# B&R Automation Studio project Soiled_PLC (part 19)

#### Main.st - Init, cyclic, exit code
```iecst
//V2.00.1 -- First stable release
//V2.00.2 -- Set brake control to be optional - This means changing when we encode the paramater structure.
//V2.00.3 -- Add new constant to set MAX_FREQUENCY
//V2.00.4 -- If the drive started not on remote it wouldn;t always go into config to start. ADD new mode for when module ok is false.
//V2.00.5 -- Add test mode for simulation
//V2.00.6 -- BUG FIX -- Minumum speed was being set to Max which stopped speed control
//V2.00.7 -- REMOVE -- Remove the old structure for settings via http
//V2.00.8 -- FIX -- Correct the scaling of MaxCurrent from settings - we now us 200 = 2A
PROGRAM _INIT
	FOR n := 1 TO MAX_DRIVES DO
		drive ACCESS ADR(ABB_EPL.Drives[n]);
		drive.Cmd.Node := 100 + n; //Set node here for now, may move to belt task
		drive.Comm.State := ABB_CONFIG;
		drive.Config.currentParam := 1; //Reset starting parameter index
	END_FOR;
END_PROGRAM

PROGRAM _CYCLIC

	FOR n := 1 TO MAX_DRIVES DO
		IF (testDrive > 0) THEN
			drive ACCESS ADR(ABB_EPL.Drives[testDrive]);
		ELSE
			drive ACCESS ADR(ABB_EPL.Drives[n]);
		END_IF;

		//Control Word												Status Word
		//Bit 0		Switch On										Bit 0	Ready To Switch On
		//Bit 1		Enable Voltage									Bit 1	Switched On
		//Bit 2		Quick Stop										Bit 2	Operation Enabled
		//Bit 3		Enable Operation								Bit 3	Fault
		//Bit 4		Not Used In Scalor Mode							Bit 4	Voltage Enabled
		//Bit 5		Not Used In Scalor Mode							Bit 5	Quick Stop
		//Bit 6		Not Used In Scalor Mode							Bit 6	Switch On Disabled
		//Bit 7		Fault Reset										Bit 7 	Warning
		//Bit 8		Halt											Bit 8	Drive Specific TBC
		//Bit 9		Operation Mode Specific							Bit 9	Remote
		//Bit 10	Reserved	??Remote Control??					Bit 10	Target Reached
		//Bit 11	Drive Specific	TBC								Bit 11 	Internal Limit Reached
		//Bit 12	Drive Specific	TBC								Bit 12	Not Used In Scalor Mode
		//Bit 13	Drive Specific	TBC								Bit 13	Not Used In Scalor Mode
		//Bit 14	Drive Specific	TBC								Bit 14	Drive Specific TBC
		//Bit 15	Drive Specific	TBC								Bit 15	Drive Specific TBC

		//Use a local instance of controlword so we don't pass changing data to the drive while processing

		controlWord := SHUT_DOWN;	// 0000 0000 0111 0110

		//Encode the controlword and statusword
		abb_packData(pData := ADR(drive));
		IF TestSystem AND NOT drive.Comm.ModuleOk THEN // TEST MODE
			IF drive.Cmd.Run THEN
				drive.Comm.State := ABB_RUNNING;
			ELSE
				drive.Status.ReadyToRun := 1;
			END_IF;
		ELSIF NOT drive.Comm.ModuleOk THEN
			drive.Comm.State := ABB_DISCONNECTED;
		ELSIF (drive.Config.params[MAX_PARAMS].status <> 0) OR (drive.Config.currentParam < MAX_PARAMS) THEN
			drive.Comm.State := ABB_CONFIG;
		ELSIF NOT drive.Status.OnRemote THEN
			drive.Comm.State := ABB_OFF_REMOTE;
		ELSIF drive.Status.Tripped THEN
			drive.Comm.State := ABB_TRIPPED;
		ELSIF NOT drive.Cmd.QuickStop THEN	//Enable quick stop
			drive.Comm.State := ABB_QUICK_STOP;
		ELSIF drive.Status.SwitchOnInhibit THEN
			drive.Comm.State := ABB_SWITCH_ON_INHIBITED;
		ELSIF drive.Comm.ErrorCode = ABB_FAULT_STO THEN
			drive.Comm.State := ABB_STO;
		END_IF;

		CASE drive.Comm.State OF

			ABB_DISCONNECTED:
				drive.Config.currentParam := 1; // Force write of parameters

			ABB_CONFIG: //Wait for module OK to be TRUE
				_setParameters; //Write params
				IF drive.Comm.ModuleOk AND (drive.Config.params[MAX_PARAMS].status = 0) THEN
					drive.Comm.State := ABB_SWITCH_ON_INHIBITED;
				END_IF;

			ABB_SWITCH_ON_INHIBITED:	//Wait for quick stop and enable to be true
				IF NOT drive.Status.SwitchOnInhibit THEN
					drive.Comm.State := ABB_NOT_READY_TO_SWITCH_ON;
				END_IF;

			ABB_NOT_READY_TO_SWITCH_ON:
				IF drive.Status.ReadyToSwitchOn THEN
					drive.Comm.State := ABB_READY_TO_SWITCH_ON;
				END_IF;

			ABB_READY_TO_SWITCH_ON:
				controlWord := SWITCH_ON; //0000 0111 0111
				IF drive.Status.ReadyToRun THEN
					drive.Comm.State := ABB_READY_TO_RUN;
				END_IF;

			ABB_READY_TO_RUN:
				controlWord := SWITCH_ON; //0000 0111 0111
				IF drive.Cmd.Run AND (ABS(drive.Cmd.TargetVelocity) >= ABB_MIN_VELOCITY) THEN	//Check min frequency is met
					drive.Comm.State := ABB_RUNNING;
				END_IF;

			ABB_RUNNING:
				controlWord := ENABLE_OPERATION; //0000 0111 1111

				IF NOT drive.Cmd.Run THEN
					drive.Comm.State := ABB_RAMP_DOWN;
				END_IF;

			ABB_RAMP_DOWN:
				controlWord := RAMP_DOWN; //0001 0111 1111
				IF drive.Comm.StatusWord.11 = 0 AND drive.Comm.ActVelocity = 0 THEN
					drive.Comm.State := ABB_READY_TO_RUN;
				END_IF;

			ABB_QUICK_STOP:
				controlWord := QUICK_STOP; //0000 0111 0010
				IF drive.Comm.StatusWord.11 = 0 AND drive.Comm.ActVelocity = 0 AND drive.Cmd.QuickStop THEN
					drive.Comm.State := ABB_READY_TO_RUN;
				END_IF;

			ABB_TRIPPED:
				//We must wait for the drive to be ready for reset and give an edge..
				controlWord := DISABLE_VOLTAGE; //0000 0000 0000
				IF drive.Comm.StatusWord.11 = 0 AND drive.Comm.ActVelocity = 0 AND NOT drive.Cmd.Reset THEN //Toggle reset to generate edge
					controlWord := FAULT_RESET;
					drive.Cmd.Reset := TRUE;
				ELSE
					drive.Cmd.Reset := FALSE;
				END_IF;
				//We can auto reset here..but we should log an error somewhere..
				IF NOT drive.Status.Tripped THEN
					drive.Comm.State := ABB_SWITCH_ON_INHIBITED;
				END_IF;

			ABB_OFF_REMOTE:
				//Remote control not active
				controlWord := SET_REMOTE;
			////				IF drive.Status.OnRemote THEN
			////					IF (drive.Config.params[MAX_PARAMS].status <> 0) THEN
			////						drive.Comm.State := ABB_CONFIG;
			////					ELSE
			////						drive.Comm.State := ABB_SWITCH_ON_INHIBITED;
			////					END_IF;
			////				END_IF;
			//				IF NOT Std.Drives_AllowLocalMode AND (drive.Config.params[13].data = Std.Drives_AllowLocalMode) THEN //Only reset the parameters if the local control mode has chnaged
			//					_encodeParameters;
			//					drive.Config.currentParam := 1; //Reset starting parameter index
			//				END_IF;
			//
			ABB_STO:
				IF drive.Comm.ErrorCode <> ABB_FAULT_STO THEN
					drive.Comm.State := ABB_SWITCH_ON_INHIBITED;
				END_IF;
		END_CASE;
		drive.Status.Running := (drive.Comm.State =  ABB_RUNNING);
		drive.Comm.ControlWord := controlWord;
	END_FOR;

	//Temp code so that we can set a node number, The NODE must already be set to 1 (DEFAULT)
	IF (newNode > 0) THEN
		setNodeNumber.enable := 1;
		setNodeNumber.node := 1;
		setNodeNumber.index := 16#4033;
		setNodeNumber.subindex := 16#03;
		setNodeNumber.pData :=  ADR(newNode);
		setNodeNumber.datalen := 2;
		setNodeNumber();
		IF (setNodeNumber.status = ERR_OK) THEN
			newNode := 0;
		END_IF;
	ELSIF saveNewNode THEN
		saveVar := 1;
		setNodeNumber.enable := 1;
		setNodeNumber.node := 1;
		setNodeNumber.index := 16#4033;
		setNodeNumber.subindex := 16#1B;
		setNodeNumber.pData :=  ADR(saveVar);
		setNodeNumber.datalen := 2;
		setNodeNumber();
		IF (setNodeNumber.status = ERR_OK) THEN
			saveNewNode := 0;
		END_IF;
	ELSIF (factoryReset > 0) THEN
		saveVar := 34560;
		setNodeNumber.enable := 1;
		setNodeNumber.node := UINT_TO_USINT(factoryReset);
		setNodeNumber.index := 16#4060;
		setNodeNumber.subindex := 16#06;
		setNodeNumber.pData :=  ADR(saveVar);
		setNodeNumber.datalen := 2;
		setNodeNumber();
		IF (setNodeNumber.status = ERR_OK) THEN
			factoryReset := 0;
		END_IF;
	END_IF;

END_PROGRAM
```

#### Types.typ - Local data types
```iecst
TYPE
	state_enum :
		(
		SLOW := 0,
		FAST := 1,
		ACC := 2,
		DEC := 3,
		MAXCURRENT := 4
		);
	BackUp : 	STRUCT
		filePath : STRING[15];
		fileDevice : STRING[10];
		status : UINT;
		ident : UDINT;
		step : backUp_enum;
		functions : backUp_functions;
	END_STRUCT;
	backUp_enum :
		(
		backUpStart := 0,
		backUpOpen := 1,
		backUpCreate := 2,
		backUpWrite := 3,
		backUpRead := 4,
		backUpClose := 5,
		backUpErrorRead := 6,
		backUpErrorWrite := 7,
		backUpExit := 100
		);
	backUp_functions : 	STRUCT
		fWrite : FileWrite;
		fRead : FileRead;
		fOpen : FileOpen;
		fCreate : FileCreate;
		fClose : FileClose;
	END_STRUCT;
END_TYPE
```

#### Variables.var - Local variables
```iecst
VAR
	abb_packData : ABB_PackData; (*Decodes status word and encodes some parameters*)
	drive : REFERENCE TO ABB_EPL_typ; (*ref var to drive structure*)
	controlWord : UINT; (*control word for drive*)
	n : USINT; (*used to hold loop state*)
	write : REFERENCE TO ABB_EPL_Param_Write_typ; (*ref var to write structutre within drive structure*)
	testDrive : UINT; (*set this to drive number you want to test*)
	i : USINT;
	state : state_enum;
	count : USINT;
	test : UINT;
	newNode : UINT;
	saveNewNode : BOOL;
	saveVar : UINT;
	factoryReset : UINT;
	setNodeNumber : EplSDOWrite;
END_VAR
```

#### encodeParameters.st
```iecst
//-----------------------------------------
//--AsEPL library Status Error Codes-------
//-----------------------------------------

//Error									Description
//0  										No error
//65534  								Function block parameter "enable" not equal to 1
//65535  								Function block still working

//31340  								Basis of error numbers, internal error
//31341  								Specified device not a POWERLINK interface
//31342  								Function can only be executed on an MN (managing node).
//31343  								Function can only be executed on a CN (controlled node).
//31344  								Read or write access failed. See errorinfo for the precise cause of the error.
//31345  								Input parameters outside of permitted value range
//31346  								Specified index already exists
//31347  								Specified subindex already exists
//31348  								Specified index does not exist
//31349  								Specified subindex does not exist
//31392  								Null pointer given as data buffer
//31399  								Error code for non-implemented functionality

//-----------------------------------------
//-----AsEPL library Error Info Codes------
//-----------------------------------------

//Error									Description
//16#0504_0000 					SDO communication timeout.
//16#0504_0001 					Invalid or unknown client/server command.
//16#0504_0002 					Size of transferred data invalid.
//16#0504_0003 					Error in sequence layer.
//16#0504_0005 					Could not allocate enough memory.
//16#0601_0000 					Cannot access object.
//16#0601_0001 					Attempted to read a write-only object.
//16#0601_0002 					Attempted to write a read-only object.
//16#0602_0000 					Object not in object dictionary.
//16#0604_0041 					Attempted to map an object in the PDO that doesn't support it.
//16#0604_0042 					Assignment would exceed PDO length.
//16#0604_0043 					General parameter incompatibility.
//16#0604_0047 					General device incompatibility.
//16#0606_0000 					Access failed due to hardware error.
//16#0607_0010 					Data type doesn't match the length of the access.
//16#0607_0012 					Length of the access is larger than the length of the data type.
//16#0607_0013 					Length of the access is smaller than the length of the data type.
//16#0609_0011 					Subindex does not exist.
//16#0609_0030 					Invalid value range.
//16#0609_0031 					Value too high for value range.
//16#0609_0032 					Value too low for value range.
//16#0609_0036 					Maximum value less than minimum value.
//16#0800_0000 					General error.
//16#0800_0020 					Cannot transfer or store data.
//16#0800_0021 					Data cannot be transferred or stored since it's being used locally by the device.
//16#0800_0022 					Data cannot be transferred or saved due to the device state.

ACTION _encodeParameters:
	//Clear all parameters
	FOR i:= 1 TO MAX_PARAMS DO
		//Clear stauts/error
		drive.Config.params[i].status := 1; //Set to 1 here, if not cleared when written is shows it has not been written
		drive.Config.params[i].errorInfo := 0;
	END_FOR;

	//Set all parameters
	//Brake Function
	drive.Config.params[1].index := 16#402C;	//Brake Control Enable 44.06
	drive.Config.params[1].subIndex := 16#6;
	drive.Config.params[1].data := BOOL_TO_DINT(drive.Cmd.BrakeFitted);	//Enable brake control
	drive.Config.params[1].datalen := 4;

	drive.Config.params[2].index := 16#400A;	//RO1 Source 10.24
	drive.Config.params[2].subIndex := 16#18;
	drive.Config.params[2].data := 22;	//Relay is active when brake is active
	drive.Config.params[2].datalen := 4;

	//Motor Data
	drive.Config.params[3].index := 16#4063;	//Motor Nominal Voltage 99.07
	drive.Config.params[3].subIndex := 16#7;
	drive.Config.params[3].data := 4150;	//415V
	drive.Config.params[3].datalen := 4;

	drive.Config.params[4].index := 16#4063;	//Motor Nominal Frequency 99.08
	drive.Config.params[4].subIndex := 16#8;
	drive.Config.params[4].data := 5000;	//50Hz
	drive.Config.params[4].datalen := 4;

	drive.Config.params[5].index := 16#4063;	//Motor Power Factor 99.11
	drive.Config.params[5].subIndex := 16#B;
	drive.Config.params[5].data := 80;	//0.8
	drive.Config.params[5].datalen := 4;

	drive.Config.params[6].index := 16#4063;	//Motor Control Mode 99.04
	drive.Config.params[6].subIndex := 16#4;
	drive.Config.params[6].data := 1;	//Scalor
	drive.Config.params[6].datalen := 2;

	//Limits
	drive.Config.params[7].index := 16#401E;	//Max Current 30.17
	drive.Config.params[7].subIndex := 16#11;
	drive.Config.params[7].data := 200;	//2.0A
	drive.Config.params[7].datalen := 4;

	drive.Config.params[8].index := 16#401E;	//Max Frequency 30.14
	drive.Config.params[8].subIndex := 16#E;
	drive.Config.params[8].data := MAX_FREQUENCY_HZ * 100;	//60Hz
	drive.Config.params[8].datalen := 4;

	//Fault Functions
	//	drive.Config.params[9].index := 16#401F;	//External Event 1 Source 31.01
	//	drive.Config.params[9].subIndex := 16#1;
	//	drive.Config.params[9].data := 2;	//Digital Input 1 Triggers Fault When Low
	//	drive.Config.params[9].datalen := 4;

	drive.Config.params[9].index := 16#4032;	//Comms loss function 50.02
	drive.Config.params[9].subIndex := 16#2;
	drive.Config.params[9].data := 1;	//Fault on comms loss
	drive.Config.params[9].datalen := 2;

	//Other
	drive.Config.params[10].index := 16#4014;	//External Commands 20.01
	drive.Config.params[10].subIndex := 16#1;
	drive.Config.params[10].data := 12;	//Fieldbus A Selected
	drive.Config.params[10].datalen := 2;

	drive.Config.params[11].index := 16#401C;	//Frequency Ext 1 Ref 28.11
	drive.Config.params[11].subIndex := 16#B;
	drive.Config.params[11].data := 4;	//Fieldbus A As Ref
	drive.Config.params[11].datalen := 4;

	drive.Config.params[12].index := 16#401F;	//STO Indication 31.22
	drive.Config.params[12].subIndex := 16#16;
	drive.Config.params[12].data := 3;	//Warning/Warning
	drive.Config.params[12].datalen := 2;

	drive.Config.params[13].index := 16#4013;	//Disable local mode 19.17
	drive.Config.params[13].subIndex := 16#11;
	drive.Config.params[13].data := BOOL_TO_DINT(NOT Std.Drives_AllowLocalMode);// 0 = Enabled ,1 = Locked
	drive.Config.params[13].datalen := 2;

	drive.Config.params[14].index := 16#4032;	//Comm loss time out 50.03
	drive.Config.params[14].subIndex := 16#3;
	drive.Config.params[14].data := 15;	//1 second
	drive.Config.params[14].datalen := 2;

	drive.Config.params[15].index := 16#401E;	//Min Frequency 30.13
	drive.Config.params[15].subIndex := 16#D;
	drive.Config.params[15].data := MAX_FREQUENCY_HZ * -100;
	drive.Config.params[15].datalen := 4;

END_ACTION
```

#### setParameters.st
```iecst
ACTION _setParameters:
	//V2.00.2 Encode parameters
	_encodeParameters;

	//Overwrite Max current
	IF ABB_EPL.Settings[drive.Cmd.Node-100].MaxCurrent > 0 THEN
		drive.Config.params[7].data := ABB_EPL.Settings[drive.Cmd.Node-100].MaxCurrent;
	END_IF;
	drive.Cmd.Acc_seconds := ABB_EPL.Settings[drive.Cmd.Node-100].Acc;
	drive.Cmd.Dec_seconds := ABB_EPL.Settings[drive.Cmd.Node-100].Dec;

	drive.Config.function.enable := TRUE;																	//Enable function block
	drive.Config.function.pDevice := ADR(PLK_INTERFACE);														//Set powerlink address in ABB_Driver init task
	drive.Config.function.node := drive.Cmd.Node; 															//Node number of drive, set in ABB_EPL[n].cmd.node if non standard.

	IF drive.Config.currentParam <= MAX_PARAMS THEN
		IF (drive.Config.params[drive.Config.currentParam].status > 0) THEN									//Call function only if not completed
			drive.Config.function.index := drive.Config.params[drive.Config.currentParam].index; 			//Powerlink index address
			drive.Config.function.subindex := drive.Config.params[drive.Config.currentParam].subIndex;		//Powerlink sub index address
			drive.Config.function.pData := ADR(drive.Config.params[drive.Config.currentParam].data);		//Value of data to write
			drive.Config.function.datalen := drive.Config.params[drive.Config.currentParam].datalen;		//Size of data type														//Call function
			IF (drive.Config.function.status = ERR_OK) THEN 												//Clear errors
				drive.Config.params[drive.Config.currentParam].status := 0;
				drive.Config.params[drive.Config.currentParam].errorInfo := 0;
				drive.Config.currentParam := drive.Config.currentParam + 1;
			ELSIF (drive.Config.function.status <> ERR_FUB_BUSY) AND (drive.Config.function.status <> ERR_FUB_ENABLE_FALSE) THEN //Store errors
				drive.Config.params[drive.Config.currentParam].status := drive.Config.function.status;
				drive.Config.params[drive.Config.currentParam].errorInfo := drive.Config.function.errorinfo;
				drive.Config.function.enable := FALSE;
//			ELSIF drive.Config.function.status <> 20925 THEN;//ERR_PLMGR_STATION_NOT_ACTIVE THEN  //Only skip if the devuce is active																																					//Skip if other error to stop PLC hanging in bootup
//				drive.Config.params[drive.Config.currentParam].status := drive.Config.function.status;
//				drive.Config.params[drive.Config.currentParam].errorInfo := drive.Config.function.errorinfo;
//				drive.Config.currentParam := drive.Config.currentParam + 1;
			END_IF;
			drive.Config.function();
		ELSE
			drive.Config.function.enable := FALSE;
		END_IF;
	END_IF;

	//Parameters should be loaded onto default settings.
	//to default the drive set 9606 t0 34560
	//Node ID (5103) has to be manually set

	write ACCESS ADR (drive.Parameters.Write);

	CASE drive.Cmd.MotorSize OF // Need to set these values correctly

		ABB_MOTOR_0_25KW:
			write.Motor_NominalCurrent_9906		:= 7; //0.68 A
			write.Motor_NominalPower_9910		:= 25; // 0.37 kW
			write.Motor_NominalSpeed_9909 		:= 1300;

		ABB_MOTOR_0_37KW_0_91A_1374:
			write.Motor_NominalCurrent_9906		:= 9; //0.91 A
			write.Motor_NominalPower_9910		:= 37; // 0.37 kW
			write.Motor_NominalSpeed_9909 		:= 1374;

		ABB_MOTOR_0_37KW_0_97A_1342:
			write.Motor_NominalCurrent_9906		:= 10; //0.97 A
			write.Motor_NominalPower_9910		:= 37; // 0.37 kW
			write.Motor_NominalSpeed_9909 		:= 1342;

		ABB_MOTOR_0_37KW_1_14A_1380:
			write.Motor_NominalCurrent_9906		:= 7; //1.14 A
			write.Motor_NominalPower_9910		:= 37; // 0.37 kW
			write.Motor_NominalSpeed_9909 		:= 1380;

		ABB_MOTOR_0_75KW:
			write.Motor_NominalCurrent_9906		:= 18; //1.75 A
			write.Motor_NominalPower_9910		:= 75; // 0.75 kW
			write.Motor_NominalSpeed_9909 		:= 1440;

		ABB_MOTOR_1_5KW:
			write.Motor_NominalCurrent_9906		:= 30;// 3 A?
			write.Motor_NominalPower_9910		:= 150;// 1.5kW
			write.Motor_NominalSpeed_9909 		:= 1450;

		ABB_MOTOR_2_2KW_4_75A_1450:
			write.Motor_NominalCurrent_9906		:= 48; //4.75 A
			write.Motor_NominalPower_9910		:= 220; // 2.2 kW
			write.Motor_NominalSpeed_9909 		:= 1450;

		ABB_MOTOR_3KW:
			write.Motor_NominalCurrent_9906		:= 64;
			write.Motor_NominalPower_9910		:= 300; // 3 kW
			write.Motor_NominalSpeed_9909 		:= 1456;

		ABB_MOTOR_CUSTOM: // Future  Alow Motor data to be set individaully
		//write.Motor_NominalCurrent_9906		:= 100;
		//write.Motor_NominalPower_9910			:= ;
		//write.Motor_NominalSpeed_9909 		:= 1450; //RPM
		//Over current = ??
		//Over torque = ??

	END_CASE;
END_ACTION
```

### Library Logical/ABB_EPL/ABB_EPL (IEC)
Depends on: AsEPL

#### ABB_EPL.typ
```iecst
TYPE
	ABB_Settings_typ : 	STRUCT
		Slow : INT;
		Fast : INT;
		Acc : INT; (*This is passed back as a whole number to make decoding easier. This in milli seconds and must be /1000 and cast to REAL.*)
		Dec : INT; (*This is passed back as a whole number to make decoding easier. This in milli seconds and must be /1000 and cast to REAL.*)
		MaxCurrent : DINT;
	END_STRUCT;
	ABB_EPL_Struct : 	STRUCT
		Settings : ARRAY[1..MAX_DRIVES]OF ABB_Settings_typ;
		Drives : ARRAY[1..MAX_DRIVES]OF ABB_EPL_typ;
		httpRequest : STRING[5000];
		httpResponse : ARRAY[0..4999]OF USINT;
		callBackUpWrite : BOOL;
	END_STRUCT;
	ABB_EPL_typ : 	STRUCT
		Comm : ABB_EPL_Comm_typ;
		Cmd : ABB_EPL_cmd_typ;
		Status : ABB_EPL_status_typ;
		Parameters : ABB_EPL_Param_typ;
		Config : EPL_Config;
	END_STRUCT;
	ABB_EPL_Comm_typ : 	STRUCT
		ControlWord : UINT;
		StatusWord : UINT;
		TargetVelocity : INT; (*RPM*)
		ActVelocity : INT; (*RPM*)
		ModuleOk : BOOL;
		State : ABB_EPL_Comm_State_enum;
		ActCurrent : DINT;
		ActTorque : DINT;
		ErrorCode : UINT;
	END_STRUCT;
	ABB_Motor_Size_enum :
		(
		ABB_MOTOR_0_25KW,
		ABB_MOTOR_0_37KW_0_91A_1374,
		ABB_MOTOR_0_37KW_0_97A_1342,
		ABB_MOTOR_0_37KW_1_14A_1380,
		ABB_MOTOR_0_75KW,
		ABB_MOTOR_1_5KW,
		ABB_MOTOR_2_2KW_4_75A_1450,
		ABB_MOTOR_3KW,
		ABB_MOTOR_CUSTOM
		);
	ABB_EPL_cmd_typ : 	STRUCT
		TargetVelocity : INT; (*RPM*)
		Run : BOOL;
		Reset : BOOL;
		QuickStop : BOOL;
		MotorSize : ABB_Motor_Size_enum;
		Dec_seconds : REAL; (*Decleration Time Seconds*)
		Acc_seconds : REAL; (*Acceleration Time Seconds*)
		Direction : ABB_DIRECTION_Enum;
		Node : USINT; (*Powerlink Node Address*)
		BrakeFitted : BOOL; (*Does the motor have a brake fitted*)
	END_STRUCT;
	ABB_EPL_status_typ : 	STRUCT
		ReadyToSwitchOn : BOOL;
		ReadyToRun : BOOL;
		Tripped : BOOL;
		DriveEnabled : BOOL;
		QuickstopActive : BOOL;
		SwitchOnInhibit : BOOL;
		Warning : BOOL;
		AtSpeed : BOOL; (**Drive is running at target velocity*)
		ActCurrent : DINT; (*Amps*)
		ActTorque : DINT; (*% of nominal motor torque*)
		ThermalTrip : BOOL;
		OnRemote : BOOL; (**Powerlink control is active*)
		Running : BOOL;
	END_STRUCT;
	ABB_EPL_Comm_State_enum :
		(
		ABB_DISCONNECTED,
		ABB_QUICK_STOP,
		ABB_CONFIG,
		ABB_SWITCH_ON_INHIBITED,
		ABB_NOT_READY_TO_SWITCH_ON,
		ABB_READY_TO_SWITCH_ON,
		ABB_READY_TO_RUN,
		ABB_RUNNING,
		ABB_TRIPPED,
		ABB_OFF_REMOTE, (**Drive not on remote control*)
		ABB_STO,
		ABB_RAMP_DOWN
		);
	ABB_EPL_Param_typ : 	STRUCT
		Read : ABB_EPL_Param_Read_typ;
		Write : ABB_EPL_Param_Write_typ;
	END_STRUCT;
	ABB_EPL_Param_Read_typ : 	STRUCT
		ActCurrent_0107 : DINT; (*Amps*)
		ActTorque_0110 : DINT; (*% of nominal motor torque*)
	END_STRUCT;
	ABB_EPL_Param_Write_typ : 	STRUCT
		Ramp_AccTime1_2872 : DINT;
		Ramp_DecTime1_2873 : DINT;
		Motor_NominalCurrent_9906 : DINT; (*1=1A*)
		Motor_NominalSpeed_9909 : DINT; (*Nominal Speed RPM*)
		Motor_NominalPower_9910 : DINT;
		QuickStopTime_2323 : DINT; (*Time in seconds for emergency stop*)
	END_STRUCT;
	ABB_DIRECTION_Enum :
		(
		ABB_DIRECTION_FWD,
		ABB_DIRECTION_REV
		);
	EPL_Config : 	STRUCT
		function : EplSDOWrite;
		currentParam : USINT;
		New_Member : USINT;
		params : ARRAY[0..MAX_PARAMS]OF EPL_SDO;
	END_STRUCT;
	EPL_SDO : 	STRUCT
		index : UINT;
		subIndex : USINT;
		data : DINT;
		datalen : UDINT;
		status : UINT;
		errorInfo : UDINT;
	END_STRUCT;
END_TYPE
```

#### Config.var
```iecst
VAR CONSTANT
	MAX_DRIVES : USINT := 23; (*Set to number of drives*)
	MAX_FREQUENCY_HZ : USINT := 70; (*Maximum Frequency Allowed in hz*)
	ABB_MIN_VELOCITY : USINT := 20; (*Minimum allowable speed of the drive*)
	PLK_INTERFACE : STRING[5] := 'IF3';
END_VAR
```

#### Constants.var - Exported constants
```iecst
VAR CONSTANT
	MAX_PARAMS : USINT := 15; (*Maximum number of params*)
END_VAR
(*CONTROL WORD STATES- DO NOT CHANGE*)
VAR CONSTANT
	DISABLE_VOLTAGE : UINT := 2#0000010000000000; (*Constanst for setting control word in case statement*)
	FAULT_RESET : UINT := 2#0000010011110000; (*Constanst for setting control word in case statement*)
	QUICK_STOP : UINT := 2#0000010001110000; (*Constanst for setting control word in case statement*)
	ENABLE_OPERATION : UINT := 2#0000010001111111; (*Constanst for setting control word in case statement*)
	RAMP_DOWN : UINT := 2#0000010101110111; (*Constanst for setting control word in case statement*)
	SHUT_DOWN : UINT := 2#0000010001110110; (*Constanst for setting control word in case statement*)
	SET_REMOTE : UINT := 2#0000010000000000; (*Constanst for setting control word in case statement*)
	SWITCH_ON : UINT := 2#0000010001110111; (*Constanst for setting control word in case statement*)
END_VAR
```

#### ABB_EPL.fun - Exported functions and function blocks
```iecst
FUNCTION_BLOCK ABB_PackData (**Pack the controlword and unpack the status word into ABB Structure *) (*$GROUP=User,$CAT=User,$GROUPICON=User.png,$CATICON=User.png*)
	VAR_INPUT
		pData : UDINT;
	END_VAR
	VAR
		abb : REFERENCE TO ABB_EPL_typ;
	END_VAR
END_FUNCTION_BLOCK
```

#### ABB_PackData.st
```iecst
(* *Pack the controlword and unpack the status word into ABB Structure  *)
FUNCTION_BLOCK ABB_PackData
	abb ACCESS pData;

	CASE abb.Cmd.Direction OF

		ABB_DIRECTION_FWD:
			abb.Comm.TargetVelocity :=	abb.Cmd.TargetVelocity;

		ABB_DIRECTION_REV:
			abb.Comm.TargetVelocity :=	abb.Cmd.TargetVelocity * - 1;
	END_CASE;

	//Control Word																Status Word
	//Bit 0		Switch On														Bit 0		Ready To Switch On
	//Bit 1		Enable Voltage											Bit 1		Switched On
	//Bit 2		Quick Stop													Bit 2		Operation Enabled
	//Bit 3		Enable Operation										Bit 3		Fault
	//Bit 4		Not Used In Scalor Mode							Bit 4		Voltage Enabled
	//Bit 5		Not Used In Scalor Mode							Bit 5		Quick Stop
	//Bit 6		Not Used In Scalor Mode							Bit 6		Switch On Disabled
	//Bit 7		Fault Reset													Bit 7 	Warning
	//Bit 8		Halt																Bit 8		Drive Specific TBC
	//Bit 9		Operation Mode Specific							Bit 9		Remote
	//Bit 10	Reserved	??Remote Control??				Bit 10	Target Reached
	//Bit 11	Drive Specific	TBC									Bit 11 	Internal Limit Reached
	//Bit 12	Drive Specific	TBC									Bit 12	Not Used In Scalor Mode
	//Bit 13	Drive Specific	TBC									Bit 13	Not Used In Scalor Mode
	//Bit 14	Drive Specific	TBC									Bit 14	Drive Specific TBC
	//Bit 15	Drive Specific	TBC									Bit 15	Drive Specific TBC

	abb.Status.ReadyToSwitchOn 	:= abb.Comm.StatusWord.0;
	abb.Status.ReadyToRun 		:= abb.Comm.StatusWord.1;
	abb.Comm.StatusWord.2; //Ready to ref-- not used
	abb.Status.Tripped 			:= abb.Comm.StatusWord.3;
	abb.Status.DriveEnabled 	:= abb.Comm.StatusWord.4; //the drive is enabled..
	abb.Status.QuickstopActive 	:= NOT abb.Comm.StatusWord.5; //QuickStop is not active
	abb.Status.SwitchOnInhibit 	:= abb.Comm.StatusWord.6; //We can't enable the drive....
	abb.Status.Warning 			:= abb.Comm.StatusWord.7;
	abb.Status.AtSpeed 			:= abb.Comm.StatusWord.8;
	abb.Status.OnRemote 		:= abb.Comm.StatusWord.9;

	abb.Status.ActCurrent := abb.Comm.ActCurrent;
	abb.Status.ActTorque := abb.Comm.ActTorque;

	//abb.Status.ThermalTrip := abb.Comm.DI.0;
	IF abb.Cmd.Acc_seconds = 0 THEN
		abb.Cmd.Acc_seconds  := 1.5;// 1.5 seconds by default
	END_IF;
	IF abb.Cmd.Dec_seconds = 0 THEN
		abb.Cmd.Dec_seconds := 1.5;// 1.5 seconds by default
	END_IF;

	abb.Parameters.Write.Ramp_AccTime1_2872 := REAL_TO_DINT(abb.Cmd.Acc_seconds * 1000.0);
	abb.Parameters.Write.Ramp_DecTime1_2873 := REAL_TO_DINT(abb.Cmd.Dec_seconds * 1000.0);

END_FUNCTION_BLOCK
```

Listed in the project but not available here: Logical/GlobalVariables/Data/Data.typ, Logical/GlobalVariables/Loading/Ldg_Funct/Types.typ, Logical/GlobalVariables/Loading/Ldg_Funct/Constants.var, Logical/GlobalVariables/BatchID/BatchID.typ, Logical/Sequences/10ms/Scan/zzTC2str/zztc2str.var, Logical/Sequences/10ms/Scan/zzTC2str/zztc2str.ab, Logical/Sequences/10ms/Scan/zzTC2end/zztc2end.var, Logical/Sequences/10ms/Scan/zzTC2end/zztc2end.ab, Logical/Sequences/10ms/zzStd/zzstd.var, Logical/Sequences/10ms/zzCount/zzcount.var, Logical/Sequences/10ms/zzCount/zzcount.ab, Logical/Sequences/10ms/4_spn1_ref/4_spn1Init.ab, Logical/Sequences/10ms/2_stb1/belt.var, Logical/Sequences/10ms/2_stb1/_setBeltTime.st, Logical/Sequences/10ms/3_clu_1/3_slu_1Init.ab, Logical/Sequences/10ms/4_pn/x_pn.var, Logical/Sequences/10ms/6_sdc1/6_sdc1Init.ab, Logical/Sequences/10ms/15_cbc1/7_sdc2Init.ab, Logical/Sequences/10ms/15_cbc1/7_sdc2.var, Logical/Sequences/10ms/25_cvc1/7_svc1Init.ab, Logical/Sequences/10ms/33_cp11, Logical/Sequences/10ms/40_cp4/12_sp2Init.ab, Logical/Sequences/10ms/44_cpr2/pr.var, Logical/Sequences/10ms/50_stn8_14/stnsa.var, Logical/Sequences/10ms/9_svc2/17_svc2Init.ab, Logical/Sequences/10ms/13_bson/14_bsonInit.ab, Logical/Sequences/10ms/13_bson/14_bson.var, Logical/Sequences/10ms/14_bsoff/15_bsoffInit.ab, Logical/Sequences/10ms/10_sb1_ref/2_belt1Init.ab, Logical/Sequences/10ms/33_fp1/12_sp2Init.ab, Logical/Sequences/10ms/12_PN2/x_pn.var, Logical/Sequences/10ms/14_svc4/18_svc3Init.ab, Logical/Sequences/10ms/13_spc1/13_spc1Init.ab, Logical/Sequences/10ms/16_sdc3/16_sdc3Init.ab, Logical/Sequences/10ms/27_sic1/ic.var, Logical/Sequences/10ms/26_spi1/11_spi1Init.ab, Logical/Sequences/10ms/23_spr3/pr.var, Logical/Sequences/10ms/zzIndi/zzindi.var, Logical/Sequences/10ms/zzIndi/zzindiCyclic.ab, Logical/Sequences/10ms/zzTCPIP/zztcpip.var, Logical/Sequences/10ms/zzIO/zzio.var, Logical/Sequences/10ms/zzOk/zzok.var, Logical/Sequences/10ms/zzUld_4a/zzuld_4.var, Logical/Sequences/200ms/CAN/CAN_Live/can_live.var, Logical/Sequences/200ms/CAN/CAN_Live/can_live.ab, Logical/Sequences/200ms/CAN/can_drv2/can_drv2.var, Logical/Sequences/200ms/udp_CTT, Logical/Sequences/200ms/zzClearMem, Logical/Sequences/200ms/zzTime/zztime.var, Logical/Sequences/200ms/zzTime/zztime.ab, Logical/Sequences/200ms/USB_Pmem/usb_pmem.var, Logical/Sequences/200ms/USB_Pmem/usb_pmem.ab, Logical/Sequences/200ms/zzWeigh/zzweigh.typ, Logical/ioimgcfg, Logical/a_flx_io, Logical/Data_BackUp/Data_BackUp.typ, Logical/Data_BackUp/Data_BackUp.var, Logical/Data_BackUp/zzDataStore/zzDataStore.var, Logical/Data_BackUp/DataBackUp/DataBackUp.typ, Logical/Data_BackUp/DataBackUp/DataBackUp.var, Logical/Data_BackUp/DataBackUp/DataSave.ab, Logical/Data_BackUp/DataBackUp/CopyToFileDevice.ab, Logical/Data_BackUp/DataBackUp/ReadFromFileDevice.ab, Logical/Data_BackUp/DataBackUp/DataBackUp.fun, Logical/Robo_Drive_Control/Robo_Drive.typ, Logical/Robo_Drive_Control/Robo_Drive.var, Logical/Robo_Drive_Control/FC302/FC302.typ, Logical/Robo_Drive_Control/FC302/FC302.var, Logical/Robo_Drive_Control/FC302/FC302.fun, Logical/Robo_Drive_Control/FC302/FC302_WriteParam.ab, Logical/Robo_Drive_Control/FC302/FC302_ReadSTW.ab, Logical/Robo_Drive_Control/FC302/FC302_WriteCTW.ab, Logical/Robo_Drive_Control/FC302/FC302_ReadParamTbl.ab, Logical/Robo_Drive_Control/FC302/FC302_ReadParam.ab, Logical/Robo_Drive_Control/Param_0_25kwStar1, Logical/Robo_Drive_Control/zzRoboPosnNames/zzRoboPosnNames.ab, Logical/Robo_Drive_Control/zzRoboPosnNames/zzRoboPosnNames.typ, Logical/Robo_Drive_Control/zzRoboPosnNames/zzRoboPosnNames.var, Logical/Robo_Drive_Control/zzRoboPosnNamesTest/zzRoboPosnNamesTest.ab, Logical/Robo_Drive_Control/zzRoboPosnNamesTest/zzRoboPosnNamesTest.typ, Logical/Robo_Drive_Control/zzRoboPosnNamesTest/zzRoboPosnNamesTest.var, Logical/Robo_Drive_Control/Lift_PosMonitor/Main.st, Logical/Robo_Drive_Control/Lift_PosMonitor/Types.typ, Logical/Robo_Drive_Control/Lift_PosMonitor/Variables.var, Logical/Robo_Drive_Control/Lift_v8_1/Lift.var, Logical/KanLink_A19/Supertrack_Kanlink_Constants/Supertrack_Constants.var, Logical/KanLink_A19/zz_KanlinkConfig/zz_KanlinkConfig.var, Logical/KanLink_A19/KGFramework/Pkg_KGStandard/Stat.var, Logical/KanLink_A19/KGFramework/Pkg_KGStandard/utfNames.typ, Logical/KanLink_A19/KGFramework/Pkg_KGStandard/kgbom.var, Logical/KanLink_A19/KGFramework/Pkg_KGStandard/KGstdLib/KG_Cmd.typ, Logical/KanLink_A19/KGFramework/Pkg_KGStandard/KGstdLib/Stat.typ, Logical/KanLink_A19/KGFramework/Pkg_KGStandard/KGstdLib/KGstdLib.typ, Logical/KanLink_A19/KGFramework/Pkg_KGStandard/KGstdLib/kgMachineState.typ, Logical/KanLink_A19/KGFramework/Pkg_KGStandard/KGstdLib/kgMachinetyp.typ, Logical/KanLink_A19/KGFramework/Pkg_KGStandard/KGstdLib/KG_Cmd.var, Logical/KanLink_A19/KGFramework/Pkg_KGStandard/KGstdLib/KGstdLib.var, Logical/KanLink_A19/KGFramework/Pkg_KGStandard/KGstdLib/kgMachineState.var, Logical/KanLink_A19/KGFramework/Pkg_KGStandard/KGstdLib/KGstdLib.fun, Logical/KanLink_A19/KGFramework/Pkg_KGStandard/KGstdLib/kgitoa_udint.st, Logical/KanLink_A19/KGFramework/Pkg_KGStandard/KGstdLib/kgatoi_udint.st, Logical/KanLink_A19/KGFramework/Pkg_KGStandard/KGstdLib/kgatoi_uint.st, Logical/KanLink_A19/KGFramework/Pkg_KGStandard/KGstdLib/kgInitBatchNoLong.st, Logical/KanLink_A19/KGFramework/Pkg_KGStandard/KGstdLib/kgNextBatchNoLong.st, Logical/KanLink_A19/KGFramework/Pkg_KGStandard/KGstdLib/kgGetMacAdress.st, Logical/KanLink_A19/KGFramework/Pkg_KGStandard/KGstdLib/kgGetBatchNoUnique.st, Logical/KanLink_A19/KGFramework/Pkg_KGStandard/KGstdLib/kgBatchNoToUDINT.st, Logical/KanLink_A19/KGFramework/Pkg_KGStandard/KGstdLib/kgUSINT16toGUID.st, Logical/KanLink_A19/KGFramework/Pkg_KGStandard/KGstdLib/kgGUIDtoSTRING.st, Logical/KanLink_A19/KGFramework/Pkg_KGStandard/KGstdLib/kgLogLine.st, Logical/KanLink_A19/KGFramework/Pkg_KGStandard/KGstdLib/kgArLogWrite.st, Logical/KanLink_A19/KGFramework/Pkg_KGStandard/KGstdLib/kgRBcreate.st, Logical/KanLink_A19/KGFramework/Pkg_KGStandard/KGstdLib/kgRBinsert.st, Logical/KanLink_A19/KGFramework/Pkg_KGStandard/KGstdLib/kgRBread.st, Logical/KanLink_A19/KGFramework/Pkg_KGStandard/KGstdLib/kgRBloc.st, Logical/KanLink_A19/KGFramework/Pkg_KGStandard/KGstdLib/kgGUIDisZero.st, Logical/KanLink_A19/KGFramework/Pkg_KGStandard/KGstdLib/kgRBbulkloc.st, Logical/KanLink_A19/KGFramework/Pkg_KGStandard/KGstdLib/kgGetLineNumberW3.st, Logical/KanLink_A19/KGFramework/Pkg_KGStandard/KGstdLib/kgGetMachineAdressW3.st, Logical/KanLink_A19/KGFramework/Pkg_KGStandard/KGstdLib/kgCheckDo.st, Logical/KanLink_A19/KGFramework/Pkg_KGStandard/KGstdLib/kgXOR.st, Logical/KanLink_A19/KGFramework/Pkg_KGStandard/KGstdLib/kgUnitconfREALtoDisplay.st, Logical/KanLink_A19/KGFramework/Pkg_KGStandard/KGstdLib/kgUnitconfDisplayToREAL.st, Logical/KanLink_A19/KGFramework/Pkg_KGStandard/KGstdLib/kgGetProgdata.st, Logical/KanLink_A19/KGFramework/Pkg_KGStandard/KGstdLib/kgSignalLight.st, Logical/KanLink_A19/KGFramework/Pkg_mnSystem/mnSystem/mnSystemCyclic.st, Logical/KanLink_A19/KGFramework/Pkg_mnSystem/mnSystem/mnSystemInit.st, Logical/KanLink_A19/KGFramework/Pkg_mnSystem/mnSystem/mnSystem.typ, Logical/KanLink_A19/KGFramework/Pkg_mnSystem/mnSystem/mnSystem.var, Logical/KanLink_A19/KGFramework/Pkg_mnSystem/Pkg_mnSystem.typ, Logical/KanLink_A19/KGFramework/Pkg_mnSystem/Pkg_mnSystem.var, Logical/KanLink_A19/KGFramework/Pkg_mnEth/Pkg_mnEth.typ, Logical/KanLink_A19/KGFramework/Pkg_mnEth/Pkg_mnEth.var, Logical/KanLink_A19/KGFramework/Pkg_mnEth/mnEth/mnEthCyclic.st, Logical/KanLink_A19/KGFramework/Pkg_mnEth/mnEth/mnEthInit.st, Logical/KanLink_A19/KGFramework/Pkg_mnEth/mnEth/mnEth.typ, Logical/KanLink_A19/KGFramework/Pkg_mnEth/mnEth/mnEth.var, Logical/KanLink_A19/KGFramework/Pkg_mnCnt/Pkg_mnCnt.typ, Logical/KanLink_A19/KGFramework/Pkg_mnCnt/Pkg_mnCnt.var, Logical/KanLink_A19/KGFramework/Pkg_mnCnt/mnCnt/mnCntCyclic.st, Logical/KanLink_A19/KGFramework/Pkg_mnCnt/mnCnt/mnCntInit.st, Logical/KanLink_A19/KGFramework/Pkg_mnCnt/mnCnt/mnCnt.typ, Logical/KanLink_A19/KGFramework/Pkg_mnCnt/mnCnt/mnCnt.var, Logical/KanLink_A19/KGFramework/Pkg_mnMsg/Pkg_mnMsg.typ, Logical/KanLink_A19/KGFramework/Pkg_mnMsg/Pkg_mnMsg.var, Logical/KanLink_A19/KGFramework/Pkg_mnMsg/mnMsg/mnMsgCyclic.st, Logical/KanLink_A19/KGFramework/Pkg_mnMsg/mnMsg/mnMsgInit.st, Logical/KanLink_A19/KGFramework/Pkg_mnMsg/mnMsg/mnMsg.typ, Logical/KanLink_A19/KGFramework/Pkg_mnMsg/mnMsg/mnMsg.var, Logical/KanLink_A19/KGFramework/Pkg_mnMsg/mnMsg/_actGetTxtFim.st, Logical/KanLink_A19/KGFramework/Pkg_mnMsg/mnMsg/_actGetTxtFimh.st, Logical/KanLink_A19/KGFramework/Pkg_mnMsg/mnMsg/_actGetOneTurnRB.st, Logical/KanLink_A19/KGFramework/Pkg_mnMsg/mnMsg/_actSetMsgOrMaint.st, Logical/KanLink_A19/KGFramework/Pkg_mnMsg/mnMsg/_actInsertRB.st, Logical/KanLink_A19/KGFramework/Pkg_mnMsg/mnMsg/_actInsertMsgL.st, Logical/KanLink_A19/KGFramework/Pkg_mnMsg/mnMsg/_actStatisticTextLCID.st, Logical/KanLink_A19/KGFramework/Pkg_mnMsg/mnMsg/_actLocMOD.st, Logical/KanLink_A19/KGFramework/Pkg_mnMsg/mnMsg/_actEventClassSel.st, Logical/KanLink_A19/KGFramework/Pkg_mnMsg/KGlibMsg/KGlibMsg.typ, Logical/KanLink_A19/KGFramework/Pkg_mnMsg/KGlibMsg/KGlibMsg.var, Logical/KanLink_A19/KGFramework/Pkg_mnMsg/KGlibMsg/KGlibMsg.fun, Logical/KanLink_A19/KGFramework/Pkg_mnMsg/KGlibMsg/msgBinSearchCfgList.st, Logical/KanLink_A19/KGFramework/Pkg_mnMsg/KGlibMsg/msgInsertMsgLine.st, Logical/KanLink_A19/KGFramework/Pkg_mnMsg/KGlibMsg/msgBinSearchTxtLine.st, Logical/KanLink_A19/KGFramework/Pkg_mnMsg/KGlibMsg/msgBinSearchHelpTxtLine.st, Logical/KanLink_A19/KGFramework/Pkg_mnMsg/KGlibMsg/msgReplSubStr.st, Logical/KanLink_A19/KGFramework/Pkg_mnMsg/KGlibMsg/msgNextChrPos.st, Logical/KanLink_A19/KGFramework/Pkg_mnParam/mnParam.typ, Logical/KanLink_A19/KGFramework/Pkg_mnParam/mnParam.var, Logical/KanLink_A19/KGFramework/Pkg_mnParam/mnParam/mnParamCyclic.st, Logical/KanLink_A19/KGFramework/Pkg_mnParam/mnParam/mnParamInit.st, Logical/KanLink_A19/KGFramework/Pkg_mnParam/mnParam/mnParamExit.st, Logical/KanLink_A19/KGFramework/Pkg_mnParam/mnParam/_mnParam.typ, Logical/KanLink_A19/KGFramework/Pkg_mnParam/mnParam/_mnParam.var, Logical/KanLink_A19/KGFramework/Pkg_mnParam/mnParam/_ExportContainer.st, Logical/KanLink_A19/KGFramework/Pkg_mnParam/mnParam/_ExportToc.st, Logical/KanLink_A19/KGFramework/Pkg_mnParam/mnParam/_DefActContainer.st, Logical/KanLink_A19/KGFramework/Pkg_mnParam/mnParam/_GetRights.st, Logical/KanLink_A19/KGFramework/Pkg_mnParam/mnParam/_BinSearchTxtLine.st, Logical/KanLink_A19/KGFramework/Pkg_mnParam/mnParam/_BinSearchHlpTxtLine.st, Logical/KanLink_A19/KGFramework/Pkg_mnParam/mnParam/_LimParam.st, Logical/KanLink_A19/KGFramework/Pkg_mnParam/mnParam/mnParam.fun, Logical/KanLink_A19/KGFramework/Pkg_mnParam/mnParam/_actInterfacePC.st, Logical/KanLink_A19/KGFramework/Pkg_mnParam/mnParam/_actInterfaceApplication.st, Logical/KanLink_A19/KGFramework/Pkg_mnParam/mnParam/_actFillEditNum.st, Logical/KanLink_A19/KGFramework/Pkg_mnParam/mnParam/_actFillEditStr.st, Logical/KanLink_A19/KGFramework/Pkg_mnParam/mnParam/_actFillNamelist.st, Logical/KanLink_A19/KGFramework/Pkg_mnParam/mnParam/_actImpModel.st, Logical/KanLink_A19/KGFramework/Pkg_mnParam/mnParamLib/mnParamLib.typ, Logical/KanLink_A19/KGFramework/Pkg_mnParam/mnParamLib/mnParamLib.var, Logical/KanLink_A19/KGFramework/Pkg_mnParam/mnParamLib/mnParamLib.fun, Logical/KanLink_A19/KGFramework/Pkg_mnParam/mnParamLib/mnParam_BinarySearchInNumeric.st, Logical/KanLink_A19/KGFramework/Pkg_mnParam/mnParamLib/mnParam_BinarySearchInString.st, Logical/KanLink_A19/KGFramework/Pkg_mnParam/mnParamLib/mnParam_CountLines.st, Logical/KanLink_A19/KGFramework/Pkg_mnParam/mnParamLib/mnParam_GetCsvDat.st, Logical/KanLink_A19/KGFramework/Pkg_mnParam/mnParamLib/mnParam_atodatetime.st, Logical/KanLink_A19/KGFramework/Pkg_mnParam/mnParamLib/mnParam_GetNextSubstring.st, Logical/KanLink_A19/KGFramework/Pkg_mnParam/mnParamLib/mnParam_GetContainerOfParamNum.st, Logical/KanLink_A19/KGFramework/Pkg_mnParam/mnParamLib/mnParam_GetContainerOfParamStrin.st, Logical/KanLink_A19/KGFramework/Pkg_mnParam/mnParamLib/GetArrayPV.st, Logical/KanLink_A19/KGFramework/Pkg_mnParam/mnParamLib/mnParam_WritePVNum.st, Logical/KanLink_A19/KGFramework/Pkg_mnParam/mnParamLib/mnParam_WritePVrNum.st, Logical/KanLink_A19/KGFramework/Pkg_mnParam/mnParamLib/mnParam_WritePVString.st, Logical/KanLink_A19/KGFramework/Pkg_mnParam/mnParamLib/mnParam_WriteBOM_Mem.st, Logical/KanLink_A19/KGFramework/Pkg_mnParam/mnParamLib/mnParam_WriteNewline_Mem.st, Logical/KanLink_A19/KGFramework/Pkg_mnParam/mnParamLib/mnParam_WriteCSV10_Mem.st, Logical/KanLink_A19/KGFramework/Pkg_mnParam/mnParamLib/mnParam_WriteCSV11_Mem.st, Logical/KanLink_A19/KGFramework/Pkg_mnParam/mnParamLib/mnParam_WriteCSV20_Mem.st, Logical/KanLink_A19/KGFramework/Pkg_mnParam/mnParamLib/mnParam_WriteCSV81_Mem.st, Logical/KanLink_A19/KGFramework/Pkg_mnParam/mnParamLib/mnParam_WriteCSV80_Mem.st, Logical/KanLink_A19/KGFramework/Pkg_mnParam/mnParamLib/mnParam_WriteCSV90_Mem.st, Logical/KanLink_A19/KGFramework/Pkg_mnParam/mnParamLib/mnParam_WriteCSV251_Mem.st, Logical/KanLink_A19/KGFramework/Pkg_mnParam/mnParamLib/mnParam_WriteCSV252_Mem.st, Logical/KanLink_A19/KGFramework/Pkg_mnParam/mnParamLib/mnParam_WriteCSV253_Mem.st, Logical/KanLink_A19/KGFramework/Pkg_mnParam/mnParamLib/mnParam_WriteCSV254_Mem.st, Logical/KanLink_A19/KGFramework/Pkg_mnParam/mnParamLib/mnParam_WriteCSV255_Mem.st, Logical/KanLink_A19/KGFramework/Pkg_mnParam/mnParamLib/mnParam_datetimetoa.st, Logical/KanLink_A19/KGFramework/Pkg_mnParam/mnParamLib/mnParam_datetoa.st, Logical/KanLink_A19/KGFramework/Pkg_mnTxt/Pkg_mnTxt.typ, Logical/KanLink_A19/KGFramework/Pkg_mnTxt/Pkg_mnTxt.var, Logical/KanLink_A19/KGFramework/Pkg_mnTxt/mnTxt/mnTxtCyclic.st, Logical/KanLink_A19/KGFramework/Pkg_mnTxt/mnTxt/mnTxtInit.st, Logical/KanLink_A19/KGFramework/Pkg_mnTxt/mnTxt/mnTxt.typ, Logical/KanLink_A19/KGFramework/Pkg_mnTxt/mnTxt/mnTxt.var, Logical/KanLink_A19/KGFramework/Pkg_mnTxt/mnTxt/_utfReplaceCtrl.st, Logical/KanLink_A19/KGFramework/Pkg_mnTxt/mnTxt/mnTxt.fun, Logical/KanLink_A19/KGFramework/Pkg_hlDFII/Pkg_hlDFII.typ, Logical/KanLink_A19/KGFramework/Pkg_hlDFII/Pkg_hlDFII.var, Logical/KanLink_A19/KGFramework/Pkg_hlDFII/hlDFII/hlDFIICyclic.st, Logical/KanLink_A19/KGFramework/Pkg_hlDFII/hlDFII/hlDFIIInit.st, Logical/KanLink_A19/KGFramework/Pkg_hlDFII/hlDFII/hlDFIIExit.st, Logical/KanLink_A19/KGFramework/Pkg_hlDFII/hlDFII/hlDFII.typ, Logical/KanLink_A19/KGFramework/Pkg_hlDFII/hlDFII/hlDFII.var, Logical/KanLink_A19/KGFramework/Pkg_hlDFII/hlDFII/_actReqScheduleTrack.st, Logical/KanLink_A19/KGFramework/Pkg_hlDFII/hlDFII/_actReqScheduleDFII.st, Logical/KanLink_A19/KGFramework/Pkg_hlDFII/hlDFII/_actProcCmdTrack.st, Logical/KanLink_A19/KGFramework/Pkg_hlDFII/hlDFII/_actProcCmdDFII.st, Logical/KanLink_A19/KGFramework/Pkg_hlDFII/hlDFII/_actProcSQLTrack.st, Logical/KanLink_A19/KGFramework/Pkg_hlDFII/hlDFII/_actProcSQLDFII.st, Logical/KanLink_A19/KGFramework/Pkg_hlDFII/hlDFII/_CreateConnectionString.st, Logical/KanLink_A19/KGFramework/Pkg_hlDFII/hlDFII/hlDFII.fun, Logical/KanLink_A19/KGFramework/Pkg_mnTest/Pkg_mnTest.typ, Logical/KanLink_A19/KGFramework/Pkg_mnTest/Pkg_mnTest.var, Logical/KanLink_A19/KGFramework/Pkg_mnTest/mnTest/mnTestCyclic.st, Logical/KanLink_A19/KGFramework/Pkg_mnTest/mnTest/mnTestInit.st, Logical/KanLink_A19/KGFramework/Pkg_mnTest/mnTest/mnTestExit.st, Logical/KanLink_A19/KGFramework/Pkg_mnTest/mnTest/mnTest.typ, Logical/KanLink_A19/KGFramework/Pkg_mnTest/mnTest/mnTest.var, Logical/KanLink_A19/KGFramework/Pkg_mnTest/mnTest/_MessageTest1.st, Logical/KanLink_A19/KGFramework/Pkg_svCPCache/Pkg_svCPCache.typ, Logical/KanLink_A19/KGFramework/Pkg_svCPCache/Pkg_svCPCache.var, Logical/KanLink_A19/KGFramework/Pkg_svCPCache/svCPCache/svCPCacheCyclic.st, Logical/KanLink_A19/KGFramework/Pkg_svCPCache/svCPCache/svCPCacheInit.st, Logical/KanLink_A19/KGFramework/Pkg_svCPCache/svCPCache/svCPCacheExit.st, Logical/KanLink_A19/KGFramework/Pkg_svCPCache/svCPCache/svCPCache.typ, Logical/KanLink_A19/KGFramework/Pkg_svCPCache/svCPCache/svCPCache.var, Logical/KanLink_A19/KGFramework/Pkg_svCPCache/svCPCache/_actCPImport.st, Logical/KanLink_A19/KGFramework/Pkg_svCPCache/svCPCache/_actIFCmd.st, Logical/KanLink_A19/KGFramework/Pkg_svCPCache/svCPCache/_actFillCPList.st, Logical/KanLink_A19/KGFramework/Pkg_svCPCache/svCPCache/_actSaveCSV.st, Logical/KanLink_A19/KGFramework/Pkg_svCPCache/svCPCache/_TrimCategory.st, Logical/KanLink_A19/KGFramework/Pkg_svCPCache/svCPCache/svCPCache.fun, Logical/KanLink_A19/KGFramework/Pkg_hlKanLink/hlKanLink.typ, Logical/KanLink_A19/KGFramework/Pkg_hlKanLink/hlKanLink.var, Logical/KanLink_A19/KGFramework/Pkg_hlKanLink/hlKanLink/KanLink.typ, Logical/KanLink_A19/KGFramework/Pkg_hlKanLink/hlKanLink/KanLinkInit.st, Logical/KanLink_A19/KGFramework/Pkg_hlKanLink/hlKanLink/KL_SaveConfDO.st, Logical/KanLink_A19/KGFramework/Pkg_hlKanLink/hlKanLink/KanLink.fun, Logical/KanLink_A19/KGFramework/Pkg_hlKanLink/KanLinkLib/CmdBI.typ, Logical/KanLink_A19/KGFramework/Pkg_hlKanLink/KanLinkLib/CmdSilo.typ, Logical/KanLink_A19/KGFramework/Pkg_hlKanLink/KanLinkLib/KanLinkLib.var, Logical/KanLink_A19/KGFramework/Pkg_hlKanLink/KanLinkLib/KLLib_CfgClient.st, Logical/KanLink_A19/KGFramework/Pkg_hlKanLink/KanLinkLib/KLLib_CfgServer.st, Logical/KanLink_A19/KGFramework/Pkg_hlKanLink/KanLinkLib/KLLib_GetPVAdr.st, Logical/KanLink_A19/KGFramework/Pkg_hlKanLink/KanLinkLib/KLLib_ReadServerPara.st, Logical/KanLink_A19/KGFramework/Pkg_hlKanLink/KanLinkLib/KLLib_InitCltPV.st, Logical/KanLink_A19/KGFramework/Pkg_hlKanLink/KanLinkLib/KLLib_ReadClientPara.st, Logical/KanLink_A19/KGFramework/Pkg_hlKanLink/KanLinkLib/KLLib_CreateStrucDef.st, Logical/KanLink_A19/KGFramework/Pkg_hlKanLink/KanLinkLib/KLLib_WriteStrucDefLine.st, Logical/KanLink_A19/KGFrameworkShare/hlDFII.Glob.var, Logical/KanLink_A19/KGFrameworkShare/mnCntGlob.var, Logical/KanLink_A19/KGFrameworkShare/mnTxtGlob.var, Logical/KanLink_A19/KGFrameworkShare/mnParamGlob.var, Logical/KanLink_A19/KGFrameworkShare/svCPCacheGlob.var, Logical/KanLink_A19/KGFrameworkShare/mnSystemGlob.var, Logical/KanLink_A19/KGFrameworkShare/Pkg_KGStandardShare/KGStandardShare.kgMsgStatus.var, Logical/KanLink_A19/KGFrameworkShare/Pkg_KGStandardShare/kgdevice.var, Logical/KanLink_A19/KGFrameworkShare/Pkg_mnEthShare/Pkg_mnEthShare.var, Logical/KanLink_A19/KGFrameworkShare/Pkg_mnMsgShare/Pkg_mnMsgShare.var, Logical/KanLink_A19/KGFrameworkShare/Pkg_hlKanLinkUser/Pkg_hlKanLinkUser.var, Logical/KanLink_A19/KGFrameworkShare/Pkg_hlKanLinkUser/KL_UserLib/Batch.typ, Logical/KanLink_A19/KGFrameworkShare/Pkg_hlKanLinkUser/KL_UserLib/KL_UserLib.typ, Logical/KanLink_A19/KGFrameworkShare/Pkg_hlKanLinkUser/KL_UserLib/KL_OnRecReq.st, Logical/KanLink_A19/KGFrameworkShare/Pkg_hlKanLinkUser/KL_UserLib/KL_UserLib.fun, Logical/KanLink_A19/KGFrameworkShare/Pkg_hlKanLinkUser/KL_UserLib/CmdWetExt.typ, Logical/KanLink_A19/KGFrameworkShare/Pkg_mnTestUser/libTestUse/libTest.typ, Logical/KanLink_A19/KGFrameworkShare/Pkg_mnTestUser/libTestUse/libTestUse.typ, Logical/KanLink_A19/KGFrameworkShare/Pkg_mnTestUser/libTestUse/libTest.var, Logical/KanLink_A19/KGFrameworkShare/Pkg_mnTestUser/libTestUse/libTestUse.var, Logical/KanLink_A19/KGFrameworkShare/Pkg_mnTestUser/libTestUse/TestUser_StopTask.st, Logical/KanLink_A19/KGFrameworkShare/Pkg_mnTestUser/libTestUse/TestUser_SetMode.st, Logical/KanLink_A19/KGFrameworkShare/Pkg_mnTestUser/libTestUse/TestUser_RunTest.st, Logical/KanLink_A19/KGFrameworkShare/Pkg_mnTestUser/libTestUse/libTestUse.fun, Logical/KanLink_A19/KGFrameworkShare/Pkg_mnTestUser/mnTestUser/mnTestUserCyclic.st, Logical/KanLink_A19/KGFrameworkShare/Pkg_mnTestUser/mnTestUser/mnTestUserInit.st, Logical/KanLink_A19/KGFrameworkShare/Pkg_mnTestUser/mnTestUser/mnTestUserExit.st, Logical/KanLink_A19/KGFrameworkShare/Pkg_mnTestUser/mnTestUser/mnTestUser.typ, Logical/KanLink_A19/KGFrameworkShare/Pkg_mnTestUser/mnTestUser/mnTestUser.var, Logical/SQL/SQLReadWriteTest/SQLSpeedTestCyclic.ab, Logical/SQL/SQLReadWriteTest/SQLSpeedTest.typ, Logical/SQL/SQLReadWriteTest/SQLSpeedTest.var, Logical/SQL/Test_bagMaint/Test_bagMaint.ab, Logical/SQL/Test_bagMaint/Test_bagMaint.var, Logical/SQL/zzGetNamesSQL/zzGetNameSQL.typ, Logical/SQL/zzGetNamesSQL/zzGetNameSQL.var, Logical/SQL/zzSQL_Lib/zzSQL_Lib.typ, Logical/SQL/zzSQL_Lib/zzSQL_Lib.var, Logical/SQL/zzSQL_Lib/Constants.var, Logical/SQL/zzSQL_Lib/zzSQL_Lib.fun, Logical/SQL/zzSQL_Lib/SQL_Write.ab, Logical/SQL/zzSQL_Lib/SQL_Read_Write.ab, Logical/SQL/zzSQLDriver/zzSQLDriver.ab, Logical/SQL/zzSQLDriver/zzSQLDriver.typ, Logical/SQL/zzSQLDriver/zzSQLDriver.var, Logical/SQL/zzTvText/zzTvText.ab, Logical/SQL/zzTvText/zzTvText.typ, Logical/SQL/zzTvText/zzTvText.var, Logical/BaseStandards/Incline/ic/ic.var, Logical/BaseStandards/On_Offgoing/x_pn/x_pn.var, Logical/BaseStandards/On_Offgoing/13_spf2/5_spf1Init.ab, Logical/BaseStandards/On_Offgoing/13_spf2/5_spf1.var, Logical/BaseStandards/Pneumatic/pc/pc.var, Logical/BaseStandards/Pneumatic/pic/pic.var, Logical/BaseStandards/36_cic6, Logical/BaseStandards/42_cp1, Logical/OPCuA/OPCuA_BagEncode/Types.typ, Logical/OPCuA/OPCuA_Displays/Types.typ, Logical/BlockPSU/zzBlockPSU/Types.typ, Logical/CustomLogs/zzWeighLog/zzWeighLog.typ, Logical/CustomLogs/zzModuleLog1/zzModuleLog.typ, Logical/Barcode_Readers/Examples/33_sp13/1_x_Point.typ, Logical/http_Lib/Constants.var, Logical/http_Lib/zzHttpDriver/Types.typ, Logical/http_Lib/zzHttpDriver/_ringBuffer.st, Logical/http_Lib/zzHttpDriver/_addToRing.st, Logical/http_Lib/zzHttpDriver/_orderRing.st, Logical/http_Lib/KanHttp/Types.typ, Logical/http_Lib/KanHttp/Constants.var, Logical/http_Lib/KanHttp/httpGetParameter.st, Logical/http_Lib/httpServer/_setBagDestination.st, Logical/http_Lib/httpServer/Types.typ, Logical/File_System/FileMgr/Constants.var, Logical/File_System/FileMgr/fileToDatObj.st, Logical/File_System/FileMgr/fileReadWrite.st, Logical/File_System/FileMgr/fileToMem.st, Logical/File_System/FileMgr/FileCopyFromDev.st, Logical/ExportsFromOriginal/0_sbelt/0_sbeltInit.ab, Logical/ExportsFromOriginal/1_stnsa/1_stnsaInit.ab, Logical/ExportsFromOriginal/2_belt1/2_belt1Init.ab, Logical/ExportsFromOriginal/3_slu_1/3_slu_1Init.ab, Logical/ExportsFromOriginal/5_spf1/5_spf1Init.ab, Logical/ExportsFromOriginal/6_sdc1/6_sdc1Init.ab, Logical/ExportsFromOriginal/7_sdc2/7_sdc2Init.ab, Logical/ExportsFromOriginal/8_svc1/8_svc1Init.ab, Logical/ExportsFromOriginal/9_sic1/9_sic1Init.ab, Logical/ExportsFromOriginal/10_ebt/10_ebtInit.ab, Logical/ExportsFromOriginal/11_spi1/11_spi1Init.ab, Logical/ExportsFromOriginal/11_spi1/11_spi1.var, Logical/ExportsFromOriginal/12_sp2/12_sp2Init.ab, Logical/ExportsFromOriginal/14_bson/14_bsonInit.ab, Logical/ExportsFromOriginal/15_bsoff/15_bsoffInit.ab, Logical/ExportsFromOriginal/17_svc2/17_svc2Init.ab, Logical/Safety/Safety/Types.typ, Logical/Safety/SafetyUI/SafetyUI.typ, Logical/Safety/SafetyUI/SafetyUI.fun, Logical/Safety/SafetyUI/itoahex.st, Logical/HoistLibrary/Hoist.var, Logical/ABB_EPL/ABB_EPL.var, Logical/ABB_EPL/ABBSettings/Types.typ
